FUNCTION_BLOCK PUBLIC FB_Device IMPLEMENTS I_Devices
//Base class for matrix, solenoid and PTTransducer classes
VAR_INPUT
	bDeviceEnable:BOOL; //Make the device Active
	bDeviceReset:BOOL;//Reset Error state
END_VAR
VAR_OUTPUT
    bError        : BOOL;   // True if in error
	bWarning :BOOL; //True if warning applicable
    eDeviceState  : E_ErrorState; // Summary device state
END_VAR
VAR
	hr : HRESULT;
	fbTrig:R_TRIG;
END_VAR

METHOD PUBLIC M_CyclicLogic : HRESULT
//  Check enable state
IF NOT bDeviceEnable THEN
	eDeviceState:=E_ErrorState.Disabled;
	M_CyclicLogic := S_Pending;
	RETURN;
END_IF

// Check reset 
fbTrig(CLK:=bDeviceReset);
IF fbTrig.Q THEN
	bError:=FALSE;
	bWarning:=FALSE;
	eDeviceState:=E_ErrorState.Healthy;
END_IF

// Handle state logic
IF bError THEN
	eDeviceState:=E_ErrorState.Alarm;
ELSIF bWarning THEN
        eDeviceState:=E_ErrorState.Warning;	
ELSE 
		eDeviceState:=E_ErrorState.Healthy;
END_IF

M_CyclicLogic := S_OK;
END_METHOD

END_FUNCTION_BLOCK

(* stored: Version 1.1.0.1
   POU FB_Device: Id {1bde026b-6494-4364-8556-c40b3b37b68a}, SpecialFunc None
   Method M_CyclicLogic: Id {4fdbe872-4aea-40f3-b2d6-233db8f39603} *)
